// TIA Portal V17 export
// export: Created 2025-03-05T08:02:21.4432536Z, ExportSetting WithDefaults, DisplayName Totally Integrated Automation Portal, DisplayVersion V17 Update 8, DisplayName TIA Portal Openness, DisplayVersion V17 Update 8, DisplayName TIA Portal Version Control Interface, DisplayVersion V17, DisplayName SINAMICS Startdrive Advanced, DisplayVersion V17 SP2, DisplayName SINAMICS Startdrive G110M, G120, G120C, G120D, G120P, G115D, DisplayVersion V17 SP2, DisplayName SINAMICS Startdrive G130, G150, S120, S150, SINAMICS MV, S210, DisplayVersion V17 SP2, DisplayName STEP 7 Professional, DisplayVersion V17 Update 8, DisplayName SINUMERIK ONE STEP 7 Toolbox, DisplayVersion V17 Update 12, DisplayName SINUMERIK 840D sl STEP 7 Toolbox, DisplayVersion V17 Update 12, DisplayName STEP 7 Safety, DisplayVersion V17 Update 6, DisplayName WinCC Advanced, DisplayVersion V17 Update 8
TYPE "SMC_JXCP1_FROM_PLC"
// stored: IsFailsafeCompliant false
   STRUCT
      STEP_NUMBER_IN_0 : Bool := false;   // STEP NUMBER BINARY DIGIT 0
      STEP_NUMBER_IN_1 : Bool := false;   // STEP NUMBER BINARY DIGIT 1
      STEP_NUMBER_IN_2 : Bool := false;   // STEP NUMBER BINARY DIGIT 2
      STEP_NUMBER_IN_3 : Bool := false;   // STEP NUMBER BINARY DIGIT 3
      STEP_NUMBER_IN_4 : Bool := false;   // STEP NUMBER BINARY DIGIT 4
      STEP_NUMBER_IN_5 : Bool := false;   // STEP NUMBER BINARY DIGIT 5
      STEP_NUMBER_UNUSED_6 : Bool := false;   // -
      STEP_NUMBER_UNUSED_7 : Bool := false;   // -
      HOLD : Bool;   // HOLD - ACTUATOR STOP
      SVON : Bool;   // SERVO ON
      DRIVE : Bool;   // DRIVE ON
      RESET : Bool;   // RESET ALARM AND OPERATION
      SETUP : Bool;   // RETURN TO ORIGIN OPERATION
      JOG_MINUS : Bool;   // JOG MINUS DIRECTION
      JOG_PLUS : Bool;   // JOG PLUS DIRECTION
      FLGTH : Bool;   // INCHING FUNCTION
      UNUSED_2_0 : Bool;   // -
      SPEED_RESTRICTION : Bool;   // SPEED RESTRICTED
      UNUSED_2_2 : Bool;   // -
      UNUSED_2_3 : Bool;   // -
      MOVEMENT_MODE : Bool;   // MOVEMENT MODE
      SPEED_BIT : Bool;   // SPEED MODE
      POSITION : Bool;   // POSITION MODE
      ACCELERATION_BIT : Bool;   // ACELERATION MODE
      DECELERATION_BIT : Bool;   // DECELERATION MODE
      PUSHING_FORCE_BIT : Bool;   // PUSHING FORCE MODE
      TRIGGER_LV_BIT : Bool;   // TRIGGER LV MODE
      PUSHING_SPEED_BIT : Bool;   // PUSHING SPEED MODE
      MOVING_FORCE_BIT : Bool;   // MOVING FORCE MODE
      AREA_1_BIT : Bool;   // AREA 1
      AREA_2_BIT : Bool;   // AREA 2
      IN_POSITION_BIT : Bool;   // IN POSITION
      START_FLAG : Bool;   // TRANSMITING NUMERICAL INSTRUCTIONS
      UNUSED_4_1 : Bool;   // -
      UNUSED_4_2 : Bool;   // -
      UNUSED_4_3 : Bool;   // -
      UNUSED_4_4 : Bool;   // -
      UNUSED_4_5 : Bool;   // -
      UNUSED_4_6 : Bool;   // -
      UNUSED_4_7 : Bool;   // -
      MOVEMENT_MODE_BIT_0 : Bool;   // MOVEMENT BIT 0 --> 1:ABS(ABSOLUTE) / 2: INC(RELATIVE)
      MOVEMENT_MODE_BIT_1 : Bool;   // MOVEMENT BIT 1 --> 1:ABS(ABSOLUTE) / 2: INC(RELATIVE)
      UNUSED_5_2 : Bool;   // -
      UNUSED_5_3 : Bool;   // -
      UNUSED_5_4 : Bool;   // -
      UNUSED_5_5 : Bool;   // -
      UNUSED_5_6 : Bool;   // -
      UNUSED_5_7 : Bool;   // -
      SPEED_VALUE : Word;   // SPEED VALUE (1mm/s)
      TARGET_POSITION : DWord;   // TARGET POSITION (0.01mm)
      ACCELERATION_VALUE : Word;   // ACCELERATION VALUE (1mm/s2)
      DECELERATION_VALUE : Word;   // DECELERATION VALUE (1mm/s2)
      PUSHING_FORCE_VALUE : Word;   // PUSHING FORCE VALUE (%)
      TRIGGER_LV_VALUE : Word;   // TRIGGER LV VALUE (%)
      PUSHING_SPEED_VALUE : Word;   // PUSHING SPEED VALEU (1mm/s)
      MOVING_FORCE_VALUE : Word;   // MOVING FORCE VALUE (%)
      AREA_1_VALUE : Word;   // AREA 1 VALUE (0.01mm)
      AREA_2_VALUE : Word;   // AREA 2 VALUE (0.01mm)
      IN_POSITION_VALUE : Word;   // IN POSITION VALUE (0.01mm)
   END_STRUCT;
END_TYPE
